PROGRAM PRG_ReplaceLongSingleCharManual
VAR
	
	sFullCode		: T_LongSTRING := 'ST=53;$02CT=10;DS=GZDNP5JOA3IL$1D;OG=3;XP=-50;YP=50;AP=-88;CS=06.2;SC=0070;QS=3;PN=1;$03$04
											ST=53;$02CT=10;DS=N7E1Y89UNK3O$1D;OG=3;XP=-50;YP=-50;AP=-88;CS=06.2;SC=0070;QS=3;PN=2;$03$04
											ST=53;$02CT=10;DS=JHWJXYFNX9DS$1D;OG=3;XP=50;YP=50;AP=-88;CS=06.2;SC=0070;QS=3;PN=3;$03$04
											ST=53;$02CT=10;DS=XGBEZLBV8A9I$1D;OG=3;XP=50;YP=-50;AP=-88;CS=06.2;SC=0070;QS=3;PN=4;$03$04'; 
	sCharRemove		: T_Char := '$1D';
	sReplacmentChar	: T_Char := '';
	
	sResult			: T_LongSTRING;
END_VAR

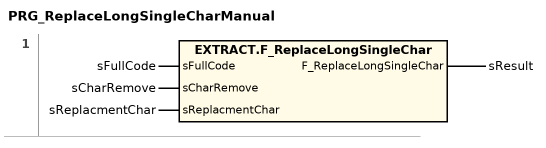
// NETWORK 1
sResult := EXTRACT.F_ReplaceLongSingleChar(sFullCode := sFullCode, sCharRemove := sCharRemove, sReplacmentChar := sReplacmentChar);

END_PROGRAM

(* stored: Version 1.1.0.1
   POU PRG_ReplaceLongSingleCharManual: Id {69fef09b-e468-4894-ae14-1661a79b2e99}, SpecialFunc None *)
